TYPE VTD_Errors_DUT :
STRUCT
	Error_Word_1:	UINT;
	Error_Word_2:	UINT;
	Error_Word_3:	UINT;
	Error_Word_4:	UINT;
	Error_Word_5:	UINT;
END_STRUCT
END_TYPE

(* stored: Version 1.1.0.1
   DUT VTD_Errors_DUT: Id {c0746d6b-55bd-4e39-82ba-70f0395478de} *)
